//{attribute 'qualified_only'}
VAR_GLOBAL
	Temperature_Transducer_A1				:	Temperature_Transducer;
	Temperature_Transducer_A1_Calibration	:	Sensor_Calibration_Multipoint;
END_VAR

(* stored: Version 1.1.0.1, ProductVersion 3.1.4024.15
   GVL GVL_Analogue_Transducer_Instruments: Id {ec551ed5-4a46-4b3b-8cfb-d86cdabacf0e} *)
